FUNCTION_BLOCK Stage2 (* Template for a Basic Function Block Type *)
  (* Standard: 61499-2 *)
  (* Version 1.0, 2021-06-20, HP *)
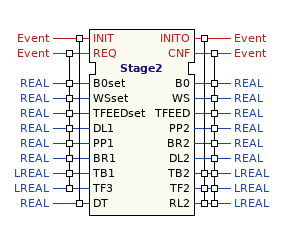
  EVENT_INPUT
    INIT WITH DT; (* Initialization Request *)
    REQ WITH B0set, WSset, TFEEDset, DL1, PP1, BR1, TB1, TF3; (* Normal Execution Request *)
  END_EVENT
  EVENT_OUTPUT
    INITO WITH TB2, TF2, RL2; (* Initialization Confirm *)
    CNF WITH TB2, DL2, TF2, BR2, PP2, RL2, WS, TFEED, B0; (* Execution Confirmation *)
  END_EVENT
  VAR_INPUT
    B0set : REAL;
    WSset : REAL;
    TFEEDset : REAL;
    DL1 : REAL;
    PP1 : REAL;
    BR1 : REAL;
    TB1 : LREAL;
    TF3 : LREAL;
    DT : REAL;
  END_VAR
  VAR_OUTPUT
    B0 : REAL;
    WS : REAL;
    TFEED : REAL;
    PP2 : REAL;
    BR2 : REAL;
    DL2 : REAL;
    TB2 : LREAL;
    TF2 : LREAL;
    RL2 : LREAL;
  END_VAR
  VAR
    AB : REAL; (* internal variabel *)
    UU : REAL;
    TREF : REAL;
    AD : REAL;
    AHC : REAL;
    AHR : REAL;
    AS : REAL;
    REC : REAL;
    WN : REAL;
    WN_1 : REAL;
    XKN : REAL;
    C1 : REAL;
    HS : REAL;
    G : REAL;
    W1 : REAL;
    TFREC : REAL;
    TS : REAL;
    DTS : REAL;
    TF2_last : REAL;
    TF3_last : REAL;
    RL2_last : REAL;
    TB2_last : REAL;
    USS : REAL;
    RHOB : REAL;
    CPB : REAL;
    CPF : REAL;
    FMW : REAL;
    HLV : REAL;
    HV : REAL;
    BPR : REAL;
    FMC : REAL;
    U : REAL;
    A : REAL;
    B : REAL;
    C : REAL;
    D1 : REAL;
    d : REAL;
    a : REAL;
    A1 : REAL;
    A2 : REAL;
    A3 : REAL;
    A4 : REAL;
    A5 : REAL;
    A6 : REAL;
    p : REAL;
    q : REAL;
    TC : REAL;
    PC : REAL;
    DTB2 : REAL;
    DEN2 : REAL;
    DH2 : REAL;
    DP2 : REAL;
    DPDH2 : REAL;
    DT2 : REAL;
    m : REAL;
    n : REAL;
    VR2 : REAL;
    DELTA2 : REAL;
    DELTA24 : REAL;
    DELTA46 : REAL;
    DELTA2_last : REAL;
    DELTA24_last : REAL;
    DELTA46_last : REAL;
  END_VAR
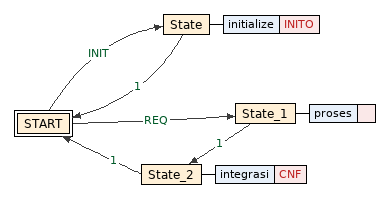
  EC_STATES
    START; (* Initial State *)
    State : initialize -> INITO;
    State_1 : proses;
    State_2 : integrasi -> CNF;
  END_STATES
  EC_TRANSITIONS
    START TO State := INIT;
    State TO START := 1;
    START TO State_1 := REQ;
    State_1 TO State_2 := 1;
    State_2 TO START := 1;
  END_TRANSITIONS
  ALGORITHM initialize IN ST: (* Initialization algorithm *)
TREF :=273.15;
AB :=57.2727;
AHC :=4069.2;
AHR :=2639.7;
AS :=3225.7;
REC :=0.0;
//TF2:=TF2;

//TFEED :=TFEED1+TREF;
 //TS:=TS1+TREF;
WN :=3.0;
XKN :=0.68;
HS:=0.11;
G :=9.81;
W1 :=0.50;

RL2 :=0.524405550;
TB2 := 361.2826497;
TF2 :=357.47363672;
TF3 := 354.9466948;

RL2_last :=RL2;
TB2_last :=TB2;
TF2_last :=TF2;
  END_ALGORITHM
  ALGORITHM proses IN ST: (* kalkulasi *)
B0 :=B0set;
WS :=WSset;
TFEED:=TFEEDset;
UU := TFEEDset;
U :=UU;

USS :=49.767;
C1 :=0.625;
RHOB :=1032.4; //maassa jenis brine
CPB :=1.00; //heatcapacity Brine
CPF :=1.00; //heat capacity feed
FMW :=23654.0;
HLV :=563.7959;
HV :=625.1971;
BPR :=2.192;
FMC :=34736.09;
//U :=UU; //feed temp



///  Calculate the physical properties

//A :=3.2437814;
//B :=5.86826*0.001;
//C :=1.1702379*0.00000001;
//D1 :=2.1878462*0.001;
//TC :=647.27;
//PC :=218.167;


A1 :=3.2437814;
A2:=5.86826*0.001;
A3:=1.1702379*0.00000001;
A4 :=2.1878462*0.001;
A5 :=647.27;
A6 :=218.167;

DTB2 :=A5-TB2;
DEN2 :=(A1+A2*DTB2+A3*DTB2*DTB2*DTB2)/(1+A4*DTB2)*DTB2/TB2;
p:=DEN2;
q:=10.0;
PP2 :=A6/(EXPT(q, p));

// calculate the brine flow rates
DP2:=PP1-PP2;
DH2:=RL2-C1*HS;
DPDH2 :=DP2*101000+G*RHOB*DH2;
m:=DPDH2*RHOB;
n:=0.5;
BR2 :=WN*XKN*RL2*(EXPT(m, n));
BR2 :=BR2*60.0/1000.0;

// calculate the vapor flow rates

DT2 :=TB2-BPR/1.8-(TF3+TF2)*0.5;
VR2 :=U*AHC*DT2/HLV/1000.0;
DL2 :=DL1+VR2;


//// state equation
DELTA2 :=(BR1-BR2-VR2)*1000.0/RHOB/AB;
DELTA24 :=((BR1*CPB*(TB1-TB2))-VR2*(HV-CPB*(TB2-TREF)))*1000.0/AB/RHOB/CPB/RL2;
DELTA46 :=((B0*CPF*(TF3-TF2)*1000+(U*AHC*DT2)))/FMW/CPF;
  END_ALGORITHM
  ALGORITHM integrasi IN ST: (* new algorithm *)
B0 :=B0set;
WS :=WSset;
TFEED:=TFEEDset;
//integrasi
RL2 := (DELTA2 + DELTA2_last)*0.5*DT + RL2_last;
DELTA2_last :=DELTA2 ;
RL2_last :=RL2;

TB2 := (DELTA24 + DELTA24_last)*0.5*DT + TB2_last;
DELTA24_last :=DELTA24 ;
TB2_last:=TB2;

TF2 := (DELTA46 + DELTA46_last)*0.5*DT + TF2_last;
DELTA46_last :=DELTA46 ;
TF2_last :=TF2;
  END_ALGORITHM
END_FUNCTION_BLOCK
